{attribute 'reflection'} 
FUNCTION_BLOCK TcLog IMPLEMENTS ILog
VAR
	{attribute 'hide'} 
	_logConditionSatisfied : BOOL; // flag that indicates, whether log condition has been satisfied.
                                // Logging will only be carried out it this evaluates to TRUE.
	{attribute 'hide'} 																
	_logDataInitialized : BOOL; // flag that indicate, whether log data has been initialized.
                             // Necessary for configuration methods to provide a fluent interface.
	{attribute 'hide'} 																
	_logData : Tc2_System.T_MaxString; // contains message to be logged.
	
	{attribute 'hide'} 
	_usedLogger : ILogCore;
	
	{attribute 'instance-path'} 
  {attribute 'noinit'} 
	_instancePath : STRING; // contains instance path
END_VAR
VAR_STAT
	_loggerSingletonInstance : ILogCore; // Wires up TcLog ("Client") to TcLogCore ("Server") (Singleton-Behaviour)
END_VAR
VAR CONSTANT
	InvalidLoggerReference : UDINT := 0;
END_VAR

// Appends any given data to the log string. Can be chained.
METHOD AppendAny : REFERENCE TO TcLog
VAR_INPUT
	Data : ANY; // Data to be appended to log string.
END_VAR
InitializeLogData();

_logData := Tc2_Standard.CONCAT(_logData, AnyToString(Data));

AppendAny REF= THIS^;
END_METHOD

// Appends a string to the log string. Can be chained.
METHOD AppendString : REFERENCE TO TcLog
VAR_INPUT
	Data : Tc2_System.T_MaxString; // Data to be appended to log string.
END_VAR
InitializeLogData();

_logData := Tc2_Standard.CONCAT(_logData, Data);
	
AppendString REF= THIS^;
END_METHOD

// Appends information about the given variable to the log string. 
// Can be chained.
// Example: 
// ---------------
// VAR
// 		myInt : INT := 10;
//		myVarInfo : __SYSTEM.VAR_INFO := __VARINFO(myInt);
// END_VAR
// Logger.AppendVariable(myVarInfo, myInt);
METHOD AppendVariable : REFERENCE TO TcLog
VAR_INPUT
	VarInfo : __SYSTEM.VAR_INFO; // VARINFO of variable to be appended to log string.
	Value : ANY; // Value of variable to be appended to log string.
END_VAR
VAR
	format : Tc2_Utilities.FB_FormatString;
	symbolName : Tc2_System.T_MaxString;
	typeName : Tc2_System.T_MaxString;
END_VAR
InitializeLogData();

symbolName := VarInfo.Symbol;
typeName := VarInfo.TypeName; 

format(
	sFormat := '%s [%s] : ',
	arg1 := Tc2_Utilities.F_STRING(symbolName),
	arg2 := Tc2_Utilities.F_STRING(typeName));
	
AppendString(format.sOut);
AppendAny(Value);

AppendVariable REF= THIS^;
END_METHOD

//	Logs the log string in DEBUG level
METHOD Debug : BOOL
VAR_INPUT
	Message : Tc2_System.T_MaxString; // Message to be appended to log string.
END_VAR
InitializeLogData();
IF _logConditionSatisfied THEN
	IF _usedLogger <> InvalidLoggerReference THEN 
		_usedLogger.LogStandardFormat(Tc2_Standard.CONCAT(_logData, Message), ShortenInstancePath(_instancePath), LogLevels.Debug); 
	ELSE
		Tc2_System.ADSLOGSTR(ADSLOG_MSGTYPE_LOG OR LogLevelToAdsLogMsgType(LogLevels.Error), 'usedLogger: No valid reference', ''); 
	END_IF
END_IF
_logDataInitialized := FALSE;
END_METHOD

// Logs the log string in ERROR level
METHOD Error : BOOL
VAR_INPUT
	Message : Tc2_System.T_MaxString; // Message to be appended to log string.
END_VAR
InitializeLogData();
IF _logConditionSatisfied THEN
	IF _usedLogger <> InvalidLoggerReference THEN 
		_usedLogger.LogStandardFormat(Tc2_Standard.CONCAT(_logData, Message), ShortenInstancePath(_instancePath), LogLevels.Error); 
	ELSE
		Tc2_System.ADSLOGSTR(ADSLOG_MSGTYPE_LOG OR LogLevelToAdsLogMsgType(LogLevels.Error), 'usedLogger: No valid reference', ''); 
	END_IF
END_IF
_logDataInitialized := FALSE;
END_METHOD

// Logs the log string in FATAL level
METHOD Fatal : BOOL
VAR_INPUT
	Message : Tc2_System.T_MaxString; // Message to be appended to log string.
END_VAR
InitializeLogData();
IF _logConditionSatisfied THEN
	IF _usedLogger <> InvalidLoggerReference THEN 
		_usedLogger.LogStandardFormat(Tc2_Standard.CONCAT(_logData, Message), ShortenInstancePath(_instancePath), LogLevels.Fatal); 
	ELSE
		Tc2_System.ADSLOGSTR(ADSLOG_MSGTYPE_LOG OR LogLevelToAdsLogMsgType(LogLevels.Error), 'usedLogger: No valid reference', ''); 
	END_IF
END_IF
_logDataInitialized := FALSE;
END_METHOD

// Logs the log string in INFORMATION level.
METHOD Information : BOOL
VAR_INPUT
	Message : Tc2_System.T_MaxString; // Message to be appended to log string.
END_VAR
InitializeLogData();
IF _logConditionSatisfied THEN
	IF _usedLogger <> InvalidLoggerReference THEN 
		_usedLogger.LogStandardFormat(Tc2_Standard.CONCAT(_logData, Message), ShortenInstancePath(_instancePath), LogLevels.Information); 
	ELSE
		Tc2_System.ADSLOGSTR(ADSLOG_MSGTYPE_LOG OR LogLevelToAdsLogMsgType(LogLevels.Error), 'usedLogger: No valid reference', ''); 
	END_IF
END_IF
_logDataInitialized := FALSE;
END_METHOD

// Initializes the reference to the core logger. Should only be called once from the core logger directly.
METHOD PUBLIC Init : BOOL
VAR_INPUT
	Ref2Core : ILogCore; // Reference to TcLoggerCore instance.
END_VAR
_loggerSingletonInstance := Ref2Core;
END_METHOD

// Necessary to provide a fluent interface of the function. 
// Has to be called at the begin of any method that returns a reference to THIS^
{attribute 'hide'}
METHOD PRIVATE InitializeLogData : BOOL
IF NOT _logDataInitialized THEN
	_logConditionSatisfied := TRUE;
	_logData := '';
	_logDataInitialized := TRUE;
	IF _usedLogger = 0 THEN _usedLogger := _loggerSingletonInstance; END_IF
END_IF
END_METHOD

// Conditional execution of the log commant. Only executes logging when Cond = TRUE.
METHOD OnCondition : REFERENCE TO TcLog
VAR_INPUT
	Cond : BOOL; // Logs data only if this condition evaluates to TRUE.
END_VAR
InitializeLogData();

_logConditionSatisfied := Cond;

OnCondition REF= THIS^;
END_METHOD

// Initializes the reference to the core logger. Should only be called once from the core logger directly.
METHOD SetLogger : BOOL
VAR_INPUT
	Ref2Core : ILogCore; // Reference to Core Logger
END_VAR
_usedLogger := Ref2Core;
END_METHOD

// Helper method. Shortens the instance path by omitting superfluent information
// such as concrete logger instance and plc/project names.
{attribute 'hide'}
METHOD PRIVATE ShortenInstancePath : Tc2_System.T_MaxString
VAR_INPUT
	Path : Tc2_System.T_MaxString; // Instance path to be shortened.
END_VAR
VAR
	i : UINT;
	shortenedPath : Tc2_System.T_MaxString;
	positionInString : INT := 0;
	positionOfLastDot : INT := 0;
END_VAR
shortenedPath := Path;

// Find last '.'
WHILE(Tc2_Standard.FIND(shortenedPath, '.') > 0) DO
	positionInString := Tc2_Standard.FIND(shortenedPath, '.');
	shortenedPath := Tc2_Standard.DELETE(shortenedPath, positionInString+1, 0);	
	positionOfLastDot := positionOfLastDot+positionInString;
END_WHILE

shortenedPath := Path;
// Delete instantiation of this FB (obvious information)
shortenedPath := Tc2_Standard.DELETE(shortenedPath, Tc2_Standard.LEN(shortenedPath)-positionOfLastDot+1, positionOfLastDot);
// Delete project information
positionInString := Tc2_Standard.FIND(shortenedPath, '.');
shortenedPath := Tc2_Standard.DELETE(shortenedPath, positionInString+1, 0);
// Delete PLC information
positionInString := Tc2_Standard.FIND(shortenedPath, '.');
shortenedPath := Tc2_Standard.DELETE(shortenedPath, positionInString+1, 0);

ShortenInstancePath := shortenedPath;
END_METHOD

// Logs directly to ADS log, ignoring the settings of the base logger.
METHOD ToAdsLog : BOOL
VAR_INPUT
	LogLevel : LogLevels; // Log level in which message should be logged to ADS.
END_VAR
InitializeLogData();

IF _logConditionSatisfied THEN
	Tc2_System.ADSLOGSTR(ADSLOG_MSGTYPE_LOG OR LogLevelToAdsLogMsgType(LogLevel), _logData, ''); 
END_IF

_logDataInitialized := FALSE;
END_METHOD

// Saves custom formatted log string. No addtitional information will be added.
METHOD ToCustomFormat : BOOL
VAR_INPUT
	Message : Tc2_System.T_MaxString; // Message to be appended to log string.
END_VAR
InitializeLogData();
IF _logConditionSatisfied THEN
	IF _usedLogger <> InvalidLoggerReference THEN 
		_usedLogger.LogCustomFormat(Tc2_Standard.CONCAT(_logData, Message)); 
	ELSE
		Tc2_System.ADSLOGSTR(ADSLOG_MSGTYPE_LOG OR LogLevelToAdsLogMsgType(LogLevels.Error), 'usedLogger: No valid reference', ''); 
	END_IF
END_IF
_logDataInitialized := FALSE;
END_METHOD

// Logs the log string in WARNING level
METHOD Warning : BOOL
VAR_INPUT
	Message : Tc2_System.T_MaxString; // Message to be appended to log string.
END_VAR
InitializeLogData();
IF _logConditionSatisfied THEN
	IF _usedLogger <> InvalidLoggerReference THEN 
		_usedLogger.LogStandardFormat(Tc2_Standard.CONCAT(_logData, Message), ShortenInstancePath(_instancePath), LogLevels.Warning); 
	ELSE
		Tc2_System.ADSLOGSTR(ADSLOG_MSGTYPE_LOG OR LogLevelToAdsLogMsgType(LogLevels.Error), 'usedLogger: No valid reference', ''); 
	END_IF
END_IF
_logDataInitialized := FALSE;
END_METHOD

END_FUNCTION_BLOCK

(* stored: Version 1.1.0.1
   POU TcLog: Id {70fb8269-5067-405b-9fff-7631f944e2d4}, SpecialFunc None
   Method AppendAny: Id {13a72111-b34b-43eb-9dd9-69ff4503fdca}
   Method AppendString: Id {7aeade46-e7f2-45b6-b46c-fff144444876}
   Method AppendVariable: Id {67339878-c4f6-4555-96b1-10fb6c84bab0}
   Method Debug: Id {a6ab730f-dade-4a97-bd0b-d6237fbafb52}
   Method Error: Id {33e3e66d-5512-4aeb-a63d-1183d4d9acad}
   Method Fatal: Id {4817ad2c-00f3-4ea2-9126-d711c8897cf3}
   Method Information: Id {ab474f28-2e54-4276-8fa1-5987c3e94a5d}
   Method Init: Id {9c7719d7-670f-46f3-92c8-88f67e360e00}
   Method InitializeLogData: Id {b4d317d9-a916-4484-9cf0-3391543593aa}
   Method OnCondition: Id {a7892907-3646-4ffc-9ebc-1cb01c1fe466}
   Method SetLogger: Id {46b10db2-eb0c-4fd5-9093-9efc1bae8abd}
   Method ShortenInstancePath: Id {b60d89ff-ac15-445d-94fa-fd767b6d287a}
   Method ToAdsLog: Id {5fabb9f2-d1d8-47fa-9304-f009c34b3048}
   Method ToCustomFormat: Id {c0ece00e-4fc1-4a0f-829f-62251f71a82e}
   Method Warning: Id {162d314a-1aa9-4cae-884b-e8b1bb3f4d70} *)
